// TIA Portal V18 export
FUNCTION "mot_speed_by_pos" : Void   // FC10, FBD
{ S7_Optimized_Access := 'TRUE' }
VERSION : 0.1
// stored: AutoNumber true, IsIECCheckEnabled false, SetENOAutomatically false, UDAEnableTagReadback false
   VAR_INPUT
      SET_SPD_DIR : Real;
      POS : Real;
      xFwdOk : Bool;
      xRevOk : Bool;
      par_fwd_limit : Real;
      par_rev_limit : Real;
      par_dist_fast : Real;
      par_speed_fast : Real;
      par_dist_crawl : Real;
      par_speed_crawl : Real;
      par_dist_stop : Real;
   END_VAR
   VAR_OUTPUT
      speed_dir : Real;
   END_VAR
   VAR_TEMP
      speed_limited_fwd : Real;
      speed_limited_rev : Real;
   END_VAR
BEGIN

REGION Network 2
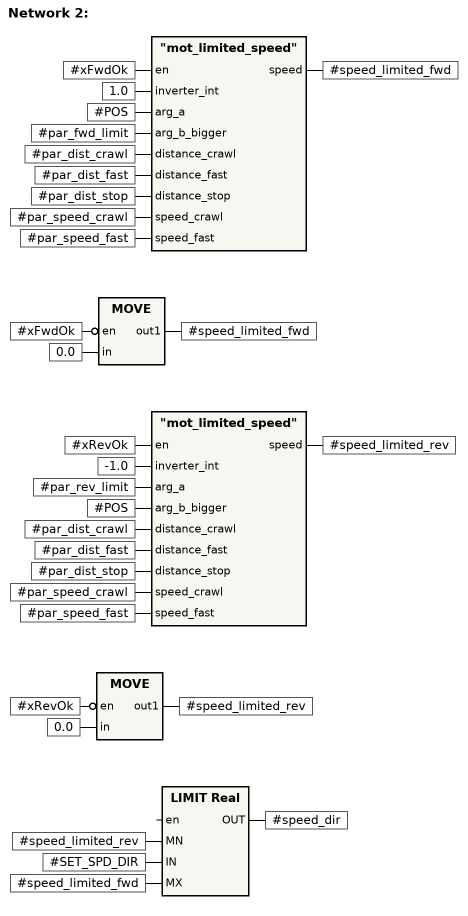
   IF #xFwdOk THEN
       "mot_limited_speed"(inverter_int := 1.0,
                           arg_a := #POS,
                           arg_b_bigger := #par_fwd_limit,
                           distance_crawl := #par_dist_crawl,
                           distance_fast := #par_dist_fast,
                           distance_stop := #par_dist_stop,
                           speed_crawl := #par_speed_crawl,
                           speed_fast := #par_speed_fast,
                           speed => #speed_limited_fwd);
   END_IF;
   IF NOT #xFwdOk THEN #speed_limited_fwd := 0.0; END_IF;
   IF #xRevOk THEN
       "mot_limited_speed"(inverter_int := -1.0,
                           arg_a := #par_rev_limit,
                           arg_b_bigger := #POS,
                           distance_crawl := #par_dist_crawl,
                           distance_fast := #par_dist_fast,
                           distance_stop := #par_dist_stop,
                           speed_crawl := #par_speed_crawl,
                           speed_fast := #par_speed_fast,
                           speed => #speed_limited_rev);
   END_IF;
   IF NOT #xRevOk THEN #speed_limited_rev := 0.0; END_IF;
   #speed_dir := LIMIT(MN := #speed_limited_rev, IN := #SET_SPD_DIR, MX := #speed_limited_fwd);
END_REGION
END_FUNCTION
